SUBAPPLICATION Uebung_226 (* Split-Bargraph: Sollwert-Eingabe treibt zwei nebeneinanderliegende Bargraphen als vorzeichenbehafteten Ausschlag *)
  (* Standard: 61499-2; Description: Copyright (c) 2026 Meisterschulen am Ostbahnhof This program and the accompanying materials are made available under the terms of the Eclipse Public License 2.0 which is available at https://www.eclipse.org/legal/epl-2.0/ SPDX-License-Identifier: EPL-2.0 *)
  (* Version 1.0, 2026-09-05, Franz Höpfinger, Meisterschulen am Ostbahnhof, initial API and implementation and/or initial documentation *)
  PACKAGE Uebungen;
  IMPORT Uebungen::const::UT::Dreieck::DefaultPool_Dreieck_BargraphSplit::Bargraph_Split_BargraphSplit;
  IMPORT Uebungen::const::UT::Dreieck::DefaultPool_Dreieck_Numeric::NumberVariable_Sollwert_N;
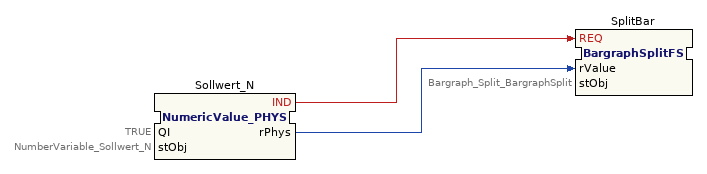
  FBS
    Sollwert_N : isobus::UT::io::NumericValue::NumericValue_PHYS(QI := TRUE, stObj := NumberVariable_Sollwert_N);
    SplitBar : isobus::UT::Q::BargraphSplitFS(stObj := Bargraph_Split_BargraphSplit);
  END_FBS
  EVENT_CONNECTIONS
    Sollwert_N.IND TO SplitBar.REQ;
  END_CONNECTIONS
  DATA_CONNECTIONS
    Sollwert_N.rPhys TO SplitBar.rValue;
  END_CONNECTIONS
END_SUBAPPLICATION
